// TIA Portal V20 export
// export: Created 2025-12-01T14:57:15.3640929Z, ExportSetting None, DisplayName Totally Integrated Automation Portal, DisplayVersion V20 Update 3, DisplayName TIA Portal Openness, DisplayVersion V20 Update 3, DisplayName TIA Portal Version Control Interface, DisplayVersion V20 Update 3, DisplayName STEP 7 Professional, DisplayVersion V20 Update 3, DisplayName STEP 7 Safety, DisplayVersion V20 Update 2, DisplayName WinCC Basic/Comfort/Advanced, DisplayVersion V20 Update 3, DisplayName WinCC Professional, DisplayVersion V20 Update 3, DisplayName WinCC Unified, DisplayVersion V20 Update 3
DATA_BLOCK "DB801_JDT01StatusCOM"   // DB801
{ S7_Optimized_Access := 'FALSE' }
AUTHOR : TRACKING
NAME : 20130301
VERSION : 3.0
// stored: AutoNumber false
   VAR
      CNTRL_OK : Bool;   // OK de la funcion AG_CNTRL
      CNTRL_Error : Bool;   // Error de la funcion AG_CNTRL
      CNTRL_PeticionActiva : Bool;   // Esta una petición Activa para la funcion AG_CNTRL
      CNTRL_Peticion : Bool;   // Realizar una petición para la función AG_CNTRL
      CNTRL_Reset : Bool;   // Petición de reset de el enlace
      Libre_005 : Bool;
      Libre_006 : Bool;
      Libre_007 : Bool;
      RecJdT_OK : Bool;   // OK de la funcion AG_RECV
      RecJdT_Error : Bool;   // Error de la funcion AG_RECV
      RecJdT_Cabecera : Bool;   // Se ha recibido la cabecera
      RecJdT_Cuerpo : Bool;   // Se ha recibido el cuerpo
      RecJdT_Reset : Bool;   // Petición de Reset de el enlace
      Libre_015 : Bool;
      Libre_016 : Bool;
      Libre_0053 : Bool;
      EmiJdT_OK : Bool;   // OK de la funcion AG_SEND
      EmiJdT_Error : Bool;   // Error de la funcion AG_SEND
      EmiJdT_PeticionActiva : Bool;   // Esta una emision activa para la funcion AG_SEND
      EmiJdT_Peticion : Bool;   // Realizar una emision para la funcion AG_SEND
      EmiJdT_Reset : Bool;   // Peticion de Reset de el enlace
      Libre_025 : Bool;
      Libre_026 : Bool;
      Libre_027 : Bool;
      EnlaceCP_OK : Bool;   // Enlace esta Activo
      EsperandoAK : Bool;   // Esperando la Confirmación del ultimo mensaje enviado
      KeepAlive_Recibido : Bool;   // Keep Alive Recibido - Hay actividad de Recepcion
      SinActividad : Bool;   // No hay actividad de Emision de Mensajes
      TMPEsperaAK_OK : Bool;   // Activado el TMP de Espera de AK - Reenvio de Mensaje
      TMPEsperaKA_OK : Bool;   // Activado el TMP de Espera de KA - Error de Comunicaciones
      TMPEnvioKA_OK : Bool;   // Activado el TMP de Envio de KA - No se han enviado ningun mensaje en X tiempo
      ResetBD : Bool;   // Limpiar toda la BD
      CNTRL_Comando : Int;   // Comando de la funcion AG_CNTRL
      CNTRL_Status : Word;   // Palabra de estado de la funcion AG_CNTRL
      CNTRL_Result01 : DWord;   // Resultado 01 de la funcion AG_CNTRL
      CNTRL_Result02 : DWord;   // Resultado 02 de la funcion AG_CNTRL
      RecJdT_Status : Word;   // Palabra de estado de la funcion AG_RECV
      RecJdT_LongitudCuerpo : UDInt;   // Numero de Bytes a recibir en el Cuerpo
      EmiJdT_Status : Word;   // Palabra de Estado de la funcion AG_SEND
      EmiJdT_Longitud : UDInt;   // Numero de bytes que hay que emitir
      ID_UltimoRecibido : UDInt;   // ID del Ultimo Mensaje Recibido
      ID_UltimoEnviado : UDInt;   // ID del Ultimo Mensaje Enviado
      TMPEsperaAK : UDInt;   // Temporizador de Espera de Confirmacion del Evento Enviado
      TMPEsperaKA : UDInt;   // Temporizador de Espera para la recepcion del Mensaje Keep Alive
      TMPEnvioKA : UDInt;   // Temporizador de Espera para el envio de el Mensaje Keep Alive
      TMPEnlace : UDInt;   // Temporizador de Espera para resetear el enlace
      TMPVisualizar : UDInt;   // Temporizador de Visualizacion de los Dispositivos
   END_VAR
BEGIN
END_DATA_BLOCK
